(* Logix 5000 project; controller axis1 vendor 1 type 14 code 155 rev 20.12; software revision 20.01 *)

TASK MainTask (continuous, watchdog 500 ms) : MainProgram

MODULES
   Local : vendor 1 type 14 code 155 (PointIO 0, rev 20.12)
      Kinetix_350 : vendor 1 type 37 code 27 (Ethernet 192.168.1.7, rev 1.1, MotionDiagnostics RPI 1 ms, MotionSync RPI 2 ms)
       : 1734-IE2V (PointIO 2, rev 3.1, Input RPI 80 ms)
      Discrete_IO : Embedded (PointIO 1, rev 20.11, Output RPI 20 ms)
       : 1734-OE2V (PointIO 3, rev 3.1, Output RPI 80 ms)
       : vendor 1 type 109 code 13 (PointIO 4, rev 3.1, Output RPI 80 ms)
END_MODULES

VAR_GLOBAL   (* controller tags *)
   Axis_1 : AXIS_CIP_DRIVE;
   Kinetix_350_Quick_Start : MOTION_GROUP;
END_VAR

PROGRAM MainProgram   (* main routine MainRoutine *)
VAR
   Axis1_Motion : MOTION_INSTRUCTION := (FLAGS := 570425344, DN := 1, STATUS := 2, STATE := 1);
   one_shot1 : BOOL;
   one_shot2 : BOOL;
END_VAR

ROUTINE MainRoutine   (* ladder *)
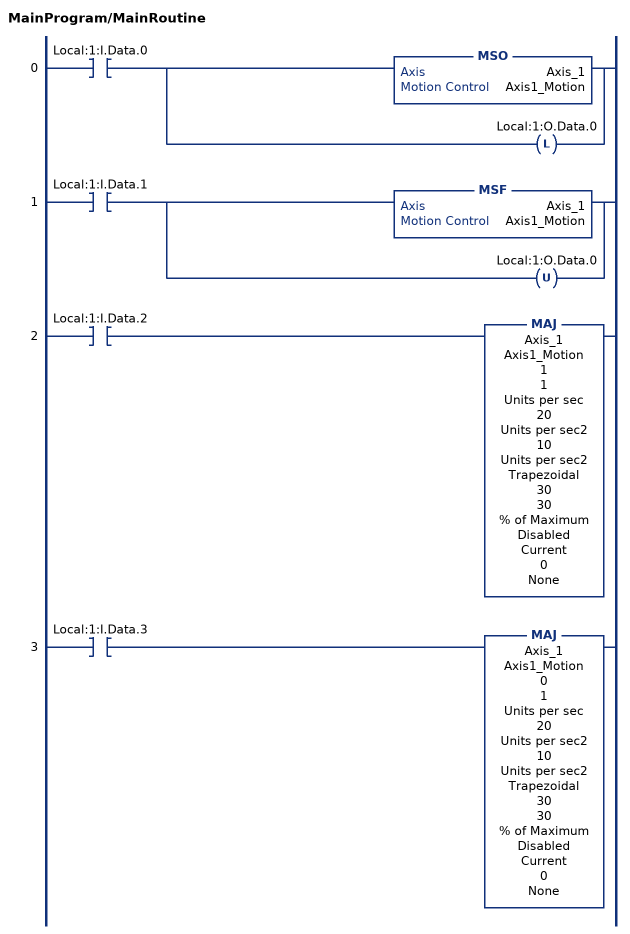
   0: XIC(Local:1:I.Data.0)[MSO(Axis_1,Axis1_Motion) ,OTL(Local:1:O.Data.0) ];
   1: XIC(Local:1:I.Data.1)[MSF(Axis_1,Axis1_Motion) ,OTU(Local:1:O.Data.0) ];
   2: XIC(Local:1:I.Data.2)MAJ(Axis_1,Axis1_Motion,1,1,Units per sec,20,Units per sec2,10,Units per sec2,Trapezoidal,30,30,% of Maximum,Disabled,Current,0,None);
   3: XIC(Local:1:I.Data.3)MAJ(Axis_1,Axis1_Motion,0,1,Units per sec,20,Units per sec2,10,Units per sec2,Trapezoidal,30,30,% of Maximum,Disabled,Current,0,None);
END_ROUTINE
END_PROGRAM
